(* IEC 61131-3 sources: my-first-repo/src, 2 files *)

(* ---- configuration.st ---- *)
CONFIGURATION MyConfiguration
    TASK Main(Priority := 1);
    PROGRAM P1 WITH Main: MyProgram;

    VAR_GLOBAL

    END_VAR
END_CONFIGURATION

(* ---- program.st ---- *)
PROGRAM MyProgram
    VAR_EXTERNAL

    END_VAR

    VAR

    END_VAR

    VAR_TEMP

    END_VAR

    myFC(iNumber:=5);
END_PROGRAM

FUNCTION myFC : Int
    VAR_INPUT
        iNumber : Int;
    END_VAR

    myFC:=iNumber;
END_FUNCTION
